Staubli VAL3: isInSafetyArea.pgx

program isInSafetyArea()
  local jointRs l_jHere
  local pointRs l_pCurrent
  local string l_sData
begin
  do
    l_pCurrent=here(flange,world)
    //**************************************************//
    //******** 用来判断机器人是否在安全工作空间 ********//
    //**************************************************//
    if (l_pCurrent.trsf.y>=nSafeMaxY or l_pCurrent.trsf.y<=nSafeMinY or l_pCurrent.trsf.x>=nSafeMaxX or l_pCurrent.trsf.x<=nSafeMinX) and _nOmacStat==3
      aioSet(aRbAlarm,10)
      call setAlarm(7)
      popUpMsg("机器人超出安全工作空间！")
      logMsg("机器人超出安全工作空间！")
      call OMAC_Abort()
    endIf

    l_sData=skToCamera
    if (l_sData=="failed")
      call setAlarm(0)
    endIf
    delay(0)
  until false
end
